INTERFACE I_StackLight

PROPERTY SystemErrorPresent : BOOL
GET
END_GET
SET
END_SET
END_PROPERTY

END_INTERFACE

(* stored: Version 1.1.0.1
   Itf I_StackLight: Id {07cbbdd6-f756-41a6-801f-a6edfbaf5f7b}
   Property SystemErrorPresent: Id {cb01a097-a4ba-4a8b-84c0-9ccc03d0df2c}
   Get Get: Id {f615aca2-3cf2-4589-8c7b-ae7660d728a9}
   Set Set: Id {c3d8a284-3b41-4b00-ab7a-11c857c780a1} *)
